MOVL C09974 V=800.0 PL=0
MOVL C09975 V=800.0 PL=0
MOVL C09976 V=800.0 PL=0
MOVL C09977 V=800.0 PL=0
MOVL C09978 V=800.0 PL=0
MOVL C09979 V=800.0 PL=0
MOVL C09980 V=800.0 PL=0
MOVL C09981 V=800.0 PL=0
MOVL C09982 V=800.0 PL=0
MOVL C09983 V=800.0 PL=0
MOVL C09984 V=800.0 PL=0
MOVL C09985 V=800.0 PL=0
MOVL C09986 V=800.0 PL=0
MOVL C09987 V=800.0 PL=0
MOVL C09988 V=800.0 PL=0
MOVL C09989 V=800.0 PL=0
MOVL C09990 V=800.0 PL=0
MOVL C09991 V=800.0 PL=0
MOVL C09992 V=800.0 PL=0
MOVL C09993 V=800.0 PL=0
MOVL C09994 V=800.0 PL=0
MOVL C09995 V=800.0 PL=0
MOVL C09996 V=800.0 PL=0
CALL JOB:A_ROOF_SIDE_0617_2_PAINT_22
END
